(* IEC 61131-3 sources: programs/VI-54/VI-54_20171205/VI-54_20171205/Stations/PLC_VI54/VI-54_171014/Class/_DriveErrorHandling, 1 file *)

(* ---- _DriveErrorHandling.st ---- *)
(*!
<Class
	Name               = "_DriveErrorHandling"
	Revision           = "1.13"
	RealtimeTask       = "false"
	CyclicTask         = "false"
	BackgroundTask     = "false"
	Sigmatek           = "true"
	OSInterface        = "false"
	HighPriority       = "false"
	Automatic          = "false"
	UpdateMode         = "Prescan"
	IconPath           = ".\Class\_DriveMngBase\Drive.ico"
	SharedCommandTable = "true"
	Objectsize         = "(540,300)"
	Comment            = "displays the error parameter of the connected Drive">
	<Channels>
		<Server Name="GetErrorInfo" Visualized="true" Initialize="false" WriteProtected="false" Retentive="false" Comment=" a write command reads the actual error state of the axis"/>
		<Server Name="I_DERROR" Visualized="true" Initialize="false" WriteProtected="true" Retentive="false" Comment="Para-Nr : 201&#13;&#10;Unit  : [-]&#13;&#10;Description : Internal Drive Errors&#13;&#13;&#10;&#13;&#13;&#10;MDD,SDD - Drives &#13;&#10;=============================================================================================&#13;&#10;Bit   1 SSI_ERROR (not supported by MDD 100)(additional Information to the Host Communication Error in [I-STATUS])&#13;&#10;Bit   2 HOST_ERROR (not supported by MDD 100)(additional Information to the Host Communication Error in [I-STATUS])&#13;&#10;Bit   3 SHORT_ERROR (short of the power stage)&#13;&#10;Bit   4 RAM_ERROR (error in the code ram area)&#13;&#10;Bit   5 FPGA_WATCHDOG_ERROR (not supported by MDD 100)(is set by the fpga watchdog mechanism)&#13;&#10;Bit   6 ADOFF_ERROR (not supported by MDD 100)(the offset of the motor current is to high)&#13;&#10;Bit   7 VCC18_ERROR (Phasing Direction Error, set when the motor turns in the wrong direction after commutation)&#13;&#10;Bit   8 VCCE_ERROR (Internal Encoder Error)&#13;&#10;Bit   9 ASMFU_IMAX_ERROR (is set if the asynchronous motor current is to high)&#13;&#10;Bit  10 PHASING_SIGNAL_STRENGTH_ERROR (Phasing Signal Strengh Error, more detailed information in Drive help parameter description I-DERROR)&#13;&#10;Bit  11 PHASING_POSITION_ERROR (is set when the position of the motor changes too drastically durin commutation)&#13;&#10;Bit  12 REGEN_ERROR (is set if the regen resistor can not be turned off)&#13;&#10;Bit  13 ENCODER_COUNTER_ERROR (not supported by MDD 100)(is set if the encoder counter check detects a fault)&#13;&#10;Bit  14 SIN_COS_COMMUT_ERROR (is set if a communication error exceeds 50ms)&#13;&#10;Bit  15 LVDS_ERROR (MDD only, is set if a communication error occurs between master and slave)&#13;&#10;Bit  16 PHASING_PHASE_SHIFT_ERROR (is set when the distance between the maximum positive/negative feedback peaks does not equal 180° +- 8°)&#13;&#10;Bit  17 PHASING_FOURIER_SIGNAL_ERROR (fourier signal cannot be calculated)&#13;&#10;&#13;&#10;DC06x&#13;&#10;=============================================================================================&#13;&#10;Bit   3 SHORT_ERROR (short of the power stage)&#13;&#10;Bit  14 FEEDBACK_ADC (feedback resolver values are not valid)(only DC061)&#13;&#10;Bit  16 SAFETY_ERROR  (safety error)&#13;&#10;Bit  17 SAFETY_WARNING (safety warning) &#13;&#10;Bit  22 Z_IMPULS_ERROR  (the z-impuls did not appeared within the time frame) (only DC062)&#13;&#10;Bit  24 FEEDBACK_SUPPLY (the feedback supply voltage fell below 15V)(only DC062)&#13;&#10;&#13;&#10;&#13;&#10;For more detailed informations, look at the parameter description of I-DERROR (201) in the Drive Help.&#13;&#13;&#10;These bits cause the Drive Error Ramp/Drive Error No Ramp in [I-STATUS]."/>
		<Server Name="I_STATUS" Visualized="true" Initialize="false" WriteProtected="true" Retentive="false" Comment="Para-Nr : 199&#13;&#10;Unit  : [-]&#13;&#10;Description : Status register:&#13;&#13;&#10;&#13;&#13;&#10;Bit  1   Mains phase (1-phase supply)&#13;&#10;Bit  2   Mains fault&#13;&#10;Bit  3   Motor axis over-current&#13;&#10;Bit  4   Over voltage DC-Link&#13;&#10;Bit  5   Under voltage DC-link&#13;&#10;Bit  6   Motor axis phase failure&#13;&#10;Bit  7   Holding brake error&#13;&#10;Bit  8   Holding brake switch damaged&#13;&#10;Bit  9   reserved&#13;&#10;Bit  10   Motor thermostat&#13;&#10;Bit 11  Ambient temperature&#13;&#10;Bit 12  Heat sink temperature&#13;&#10;Bit 13  Feedback Error&#13;&#10;Bit 14  Commutation error&#13;&#10;Bit 15  Over speed&#13;&#10;Bit 16  Contouring Error&#13;&#10;Bit 17  Trajectory Error&#13;&#10;Bit 18  Host Communication Error&#13;&#10;Bit 19  Drive Error Ramp, for additional information see [I-DERROR]&#13;&#10;Bit 20  Drive Error No Ramp, for additional information see [I-DERROR]&#13;&#10;Bit 21  External Enable Locked Error&#13;&#10;Bit 22  IGBT Driver Voltage Error&#13;&#10;Bit 23  max. Regen Power Error&#13;&#10;Bit 24  24V Brake Supply Error&#13;&#10;Bit 25  reserved&#13;&#10;Bit 26  I2T-Error&#13;&#10;Bit 27  Motor Temperature Warning&#13;&#10;Bit 28  Motor Parameter Error&#13;&#10;Bit 29  Multi-Turn Position Error&#13;&#10;Bit 30  Max Sum Power Limitation&#13;&#10;Bit 31  Speed Controler in Saturation&#13;&#10;Bit 32  Fan Error &#13;&#10;&#13;&#13;&#10;The masks  [G-MASKE1], [G-MASKE2], [G-MASKW] and [G-MASKD] &#13;&#10;define if the corresponding bit of I-STATUS causes a cast of the motor, a ramp stop of the motor, a warning or nothing.&#13;&#13;&#10;This errors can be cleared with [K-CLRF].&#13;&#10;For more detailed informations, look at the parameter description of I-STATUS(199) in the Drive Help.&#13;&#10;"/>
	</Channels>
	<RevDoku>
		<Owner Company="Sigmatek" Author="HasHan"/>
		<Dokumentation Revision="1.13" Date="08.11.2016" Author="ZoePat" Company="Sigmatek" Description="Client &quot;DriveAxis&quot; is now not required."/>
		<Dokumentation Revision="1.12" Date="03.11.2015" Author="EisMic" Company="Sigmatek" Description="Bits in server comment now start from 1 instead of 0 to be consistent with the lasal help and the type of the server.."/>
		<Dokumentation Revision="1.11" Date="16.06.2015" Author="EisMic" Company="Sigmatek" Description="Updated description from I-STATUSand I-DERROR Bits."/>
		<Dokumentation Revision="1.10" Date="04.12.2013" Author="ObeChr" Company="Sigmatek" Description="Added missing Bits in Type for Server I-STATUS + I-DERROR"/>
		<Dokumentation Revision="1.1" Date="10.08.2010" Author="Ramand" Company="Sigmatek" Description="For the number of parameters in this group now a constant is used instead of the numerical value for easier change in the future"/>
		<Dokumentation Revision="1.0" Date="05.08.2009" Author="HasHan" Company="Sigmatek" Description="Creation"/>
	</RevDoku>
	<Network Name="_DriveErrorHandling">
		<!-- List of Components in this network -->
		<Components>
			<Object
				Name       = "_base"
				Class      = "_DriveParaBase"
				Position   = "(218,120)"
				Visualized = "false">
				<Channels>
					<Server Name="State"/>
					<Client Name="DriveAxis"/>
					<Client Name="ErrorCode"/>
				</Channels>
			</Object>
		</Components>
		<Comments>
		</Comments>
		<!-- List of Connections in this network -->
		<Connections>
			<Connection Source="this.State" Destination="_base.State" Vertices="(740,210),(568,210),"/>
			<Connection Source="_base.DriveAxis" Destination="this.DriveAxis" Vertices="(218,210),(38,210),"/>
			<Connection Source="_base.ErrorCode" Destination="this.ErrorCode" Vertices="(218,270),(38,270),"/>
		</Connections>
		<!-- Headerfiles -->
		<Options>
		</Options>
	</Network>
</Class>
*)
#pragma using _DriveParaBase

_DriveErrorHandling : CLASS
: _DriveParaBase
  //Servers:
	GetErrorInfo 	: SvrCh_DINT;
	I_STATUS 	: SvrCh__SDDISTATE;
	I_DERROR 	: SvrCh__SDDIDERROR;
  //Clients:
  //Variables:
  //Functions:

	FUNCTION VIRTUAL GLOBAL Init;

	FUNCTION VIRTUAL GLOBAL RefreshPara
		VAR_INPUT
			usParaNr 	: USINT;
			dValue 	: DINT;
		END_VAR;

	FUNCTION VIRTUAL GLOBAL RefreshAllPara;

	FUNCTION GLOBAL GetErrorInformation;

	FUNCTION VIRTUAL GLOBAL GetErrorInfo::Write
		VAR_INPUT
			input (EAX) 	: DINT;
		END_VAR
		VAR_OUTPUT
			result (EAX) 	: DINT;
		END_VAR;
  //Tables:
	FUNCTION @STD
		VAR_OUTPUT
			ret_code	: CONFSTATES;
		END_VAR;
	FUNCTION GLOBAL TAB @CT_;
END_CLASS;

FUNCTION VIRTUAL GLOBAL _DriveErrorHandling::Init

  if (IsAxisConnected() = TRUE) then
    DriveAxis.AddParaObjects(Index:=IDX_ERRORHANDLING, pThis:=this); // add the object in the list of the axis
    DriveAxis := ERROR;
    State := DriveAxis.CmdState;
  end_if;

END_FUNCTION

FUNCTION VIRTUAL GLOBAL _DriveErrorHandling::GetErrorInfo::Write
	VAR_INPUT
		input (EAX) 	: DINT;
	END_VAR
	VAR_OUTPUT
		result (EAX) 	: DINT;
	END_VAR

	GetErrorInfo := input;
 	result := GetErrorInfo;
  GetErrorInformation();

END_FUNCTION

FUNCTION VIRTUAL GLOBAL _DriveErrorHandling::RefreshPara
	VAR_INPUT
		usParaNr 	: USINT;
		dValue 	: DINT;
	END_VAR

  case usParaNr of

    SDD_I_STATUS :
      I_STATUS$DINT := dValue;

    SDD_I_DERROR :
      I_DERROR$DINT := dValue;

  end_case;

END_FUNCTION

FUNCTION GLOBAL _DriveErrorHandling::GetErrorInformation

  SetASyncCmd(ParaNr:= SDD_I_STATUS, ParaRdWr:= 0, ParaValue:= 0, pThis:= this);
  SetASyncCmd(ParaNr:= SDD_I_DERROR, ParaRdWr:= 0, ParaValue:= 0, pThis:= this);

END_FUNCTION

FUNCTION VIRTUAL GLOBAL _DriveErrorHandling::RefreshAllPara

  // number of Parameters in this group
  AnzASyncPara += NBR_ERRORHANDLING;

END_FUNCTION
